Universal Robots PolyScope program: sprayFront.urp

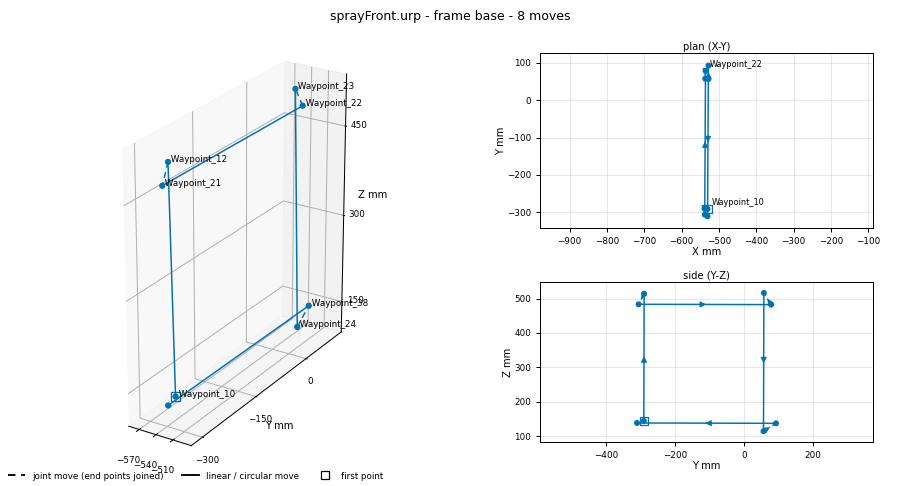
[picture p0: tool path of sprayFront.urp in frame base, 8 of 8 moves have a stored position in this frame; points joined in program order, loops and branches not executed]
Program sprayFront (installation=April22Cube directory=/programs/April2022Sand/subs createdIn=5.11.5.1010327 lastSavedIn=5.11.5.1010327 robotSerialNumber=20215500677)
Calibrated DH parameters: a=[0.000204, -0.239222, -0.391845, -0.000001, 0.000022, 0]; d=[0.162722, -355.808559, 353.37206, 2.570385, 0.099741, 0.099629]; alpha=[1.571124, 0.000988, 0.008295, 1.568963, -1.570303, 0]; deltaTheta=[0, -0.973091, 7.204745, 0.05153, 0, 0]
Robot Program (runOnlyOnce=false)
  Folder SprayFront
    MoveJ speed 60 deg/s, acceleration 80 deg/s^2 (useActiveTCP=false) tcp=SprayTCP; feature=CubeFront
      Waypoint Waypoint_10: TCP in base x=-530.531 y=-291.052 z=144.441 mm, rx=-2.2301 ry=-0.0105 rz=2.1935 rad; joints [-0.761, -65.891, 118.661, -46.487, 45.268, 89.493] deg; TCP offset x=20.839 y=-27.14 z=105.994 mm, rx=0.1226 ry=1.1769 rz=2.8697 rad; feature pose in base x=-150.564 y=-110.257 z=792.369 mm, rx=-0.0207 ry=-0.0133 rz=3.0697 rad
      Set DigitalOutput pin=SprayerOn; digitalValue=1
    MoveL speed 100 mm/s, acceleration 1200 mm/s^2 (useActiveTCP=true) feature=CubeFront
      Waypoint Waypoint_12: TCP in base x=-538.683 y=-290.104 z=513.862 mm, rx=-2.2302 ry=-0.0105 rz=2.1934 rad; joints [-0.84, -86.478, 83.393, 9.273, 44.774, 89.634] deg
      Set DigitalOutput pin=SprayerOn; digitalValue=0
      MoveDirectionNode (selectedDirection=ZMinus toolParams=0.2, 1.2) feature=Joint_6_name
        Until DISTANCE (allowActions=false deceleration=3 distanceNodeType=STOP) Distance=0.1; motionParameters(blendRadius=0)
    MoveJ speed 60 deg/s, acceleration 80 deg/s^2 (useActiveTCP=false) tcp=SprayTCP; feature=CubeFront
      Waypoint Waypoint_21: TCP in base x=-538.097 y=-306.157 z=483.391 mm, rx=1.2299 ry=-1.2185 rz=-1.2154 rad; joints [22.708, -78.928, 107.314, -73.338, 103.019, 167.126] deg; TCP offset x=20.839 y=-27.14 z=105.994 mm, rx=0.1226 ry=1.1769 rz=2.8697 rad
      Set DigitalOutput pin=SprayerOn; digitalValue=1
    MoveL speed 100 mm/s, acceleration 1200 mm/s^2 (useActiveTCP=false) tcp=SprayTCP; feature=CubeFront
      Waypoint Waypoint_22: TCP in base x=-536.01 y=78.845 z=482.449 mm, rx=1.2299 ry=-1.2184 rz=-1.2154 rad; joints [-28.836, -93.233, 123.857, -79.597, 66.516, 204.312] deg; TCP offset x=20.839 y=-27.14 z=105.994 mm, rx=0.1226 ry=1.1769 rz=2.8697 rad
      Set DigitalOutput pin=SprayerOn; digitalValue=0
      MoveDirectionNode (selectedDirection=ZMinus toolParams=0.2, 1.2) feature=Joint_6_name
        Until DISTANCE (allowActions=false deceleration=3 distanceNodeType=STOP) Distance=0.1; motionParameters(blendRadius=0)
    MoveJ speed 60 deg/s, acceleration 80 deg/s^2 (useActiveTCP=false) tcp=SprayTCP; feature=CubeFront
      Waypoint Waypoint_23: TCP in base x=-536.857 y=57.735 z=516.338 mm, rx=0.0075 ry=-1.5876 rz=-0.0151 rad; joints [-3.715, -89.488, 83.743, 1.67, 131.045, 270.018] deg; TCP offset x=20.839 y=-27.14 z=105.994 mm, rx=0.1226 ry=1.1769 rz=2.8697 rad
      Set DigitalOutput pin=SprayerOn; digitalValue=1
    MoveL speed 100 mm/s, acceleration 1200 mm/s^2 (useActiveTCP=false) tcp=SprayTCP; feature=CubeFront
      Waypoint Waypoint_24: TCP in base x=-528.032 y=56.71 z=114.659 mm, rx=0.0075 ry=-1.5874 rz=-0.0151 rad; joints [-3.717, -66.449, 123.019, -60.833, 131.469, 269.749] deg; TCP offset x=20.839 y=-27.14 z=105.994 mm, rx=0.1226 ry=1.1769 rz=2.8697 rad
      Set DigitalOutput pin=SprayerOn; digitalValue=0
      MoveDirectionNode (selectedDirection=ZMinus toolParams=0.2, 1.2) feature=Joint_6_name
        Until DISTANCE (allowActions=false deceleration=3 distanceNodeType=STOP) Distance=0.1; motionParameters(blendRadius=0)
    MoveJ speed 60 deg/s, acceleration 80 deg/s^2 (useActiveTCP=false) tcp=SprayTCP; feature=CubeFront
      Waypoint Waypoint_38: TCP in base x=-528.302 y=92.929 z=137.544 mm, rx=1.2295 ry=-1.2182 rz=-1.2157 rad; joints [-31.314, -39.364, 132.373, -142.669, 64.779, 205.918] deg
      Set DigitalOutput pin=SprayerOn; digitalValue=1
    MoveL speed 100 mm/s, acceleration 1200 mm/s^2 (useActiveTCP=false) tcp=SprayTCP; feature=CubeFront
      Waypoint Waypoint_25: TCP in base x=-530.503 y=-310.8 z=138.54 mm, rx=1.2295 ry=-1.2182 rz=-1.2157 rad; joints [23.481, -38.767, 115.153, -121.572, 103.542, 166.189] deg
      Set DigitalOutput pin=SprayerOn; digitalValue=0
      MoveDirectionNode (selectedDirection=ZMinus toolParams=0.2, 1.2) feature=Joint_6_name
        Until DISTANCE (allowActions=false deceleration=3 distanceNodeType=STOP) Distance=0.1; motionParameters(blendRadius=0)
